// TIA Portal V20 export
// export: Created 2025-12-01T14:57:11.2590179Z, ExportSetting None, DisplayName Totally Integrated Automation Portal, DisplayVersion V20 Update 3, DisplayName TIA Portal Openness, DisplayVersion V20 Update 3, DisplayName TIA Portal Version Control Interface, DisplayVersion V20 Update 3, DisplayName STEP 7 Professional, DisplayVersion V20 Update 3, DisplayName STEP 7 Safety, DisplayVersion V20 Update 2, DisplayName WinCC Basic/Comfort/Advanced, DisplayVersion V20 Update 3, DisplayName WinCC Professional, DisplayVersion V20 Update 3, DisplayName WinCC Unified, DisplayVersion V20 Update 3
FUNCTION "FC894_Obtener_ValorDeEtiqueta" : Void   // FC894, STL
TITLE = "Evento_EtiquetaValor"
{ S7_Optimized_Access := 'FALSE' }
AUTHOR : TRACKING
NAME : 20160411
VERSION : 3.4
// Convertir un texto DWORD a un valor numerico UInt
// stored: AutoNumber false
   VAR_INPUT
      EtiquetaEvento : DWord;   // Etiqueta del evento Recibido
   END_VAR
   VAR_OUTPUT
      ValorEvento : UInt;   // Valor del Evento Recibido para la BD
   END_VAR
   VAR_TEMP
      Indice : UInt;   // Indice para recorrer el array
   END_VAR
BEGIN

NETWORK
TITLE = Inicializar
// - Inicializar la salida
/////////////////////////////////////////////////////////////////////////////////////
// Inicializar la salida

      L     0;
      T     #ValorEvento;


NETWORK
TITLE = Buscar la Etiqueta para Obtner el valor
/////////////////////////////////////////////////////////////////////////////////////
/////////////////////////////////////////////////////////////////////////////////////
/////////////////////////////////////////////////////////////////////////////////////
// --- Bucle de Busqueda de Etiqueta
      L     1;
      T     #Indice;

Inicio_BucleDeBusqueda:NOP   0;
      L     "DB870_ConversorEventos".Etiqueta_A_Valor[#Indice].Etiqueta;
      L     #EtiquetaEvento;
      ==D;
      JC    Encontrada_EtiquetaBuscada;

// --- Final de Etiquetas Existentes
      L     "DB870_ConversorEventos".Etiqueta_A_Valor[#Indice].Etiqueta;
      L     0;
      ==D;
      JC    Final;  // Hay mas etiquetas?

// --- Maximo del Array de Etiquetas
      L     #Indice;
      L     "CTE_MaxArrayConversion";
      >=I;
      JC    Final;  // No se ha encontrado?


// --- Continuar la Busqueda
      L     #Indice;
      L     1;
      +I;
      T     #Indice;

      JU    Inicio_BucleDeBusqueda;

/////////////////////////////////////////////////////////////////////////////////////
/////////////////////////////////////////////////////////////////////////////////////
/////////////////////////////////////////////////////////////////////////////////////
// --- Etiqueta Encontrada
Encontrada_EtiquetaBuscada:NOP   0;
      L     "DB870_ConversorEventos".Etiqueta_A_Valor[#Indice].Valor;
      T     #ValorEvento;



NETWORK
TITLE = Final
/////////////////////////////////////////////////////////////////////////////////////
// Final de la funcion
Final:NOP   0;


END_FUNCTION
